SUBAPPLICATION Uebung_011f_AX (* Numeric Value Input I3 Durchschleifen auf N3 (Input und Output PHYS via NumericObjectPool_S) *)
  (* Standard: 61499-2; Description: Copyright (c) 2023 Meisterschulen am Ostbahnhof This program and the accompanying materials are made available under the terms of the Eclipse Public License 2.0 which is available at https://www.eclipse.org/legal/epl-2.0/ SPDX-License-Identifier: EPL-2.0 *)
  (* Version 1.0, 2026-04-14, Franz Höpfinger, Meisterschulen am Ostbahnhof, initial API and implementation and/or initial documentation *)
  PACKAGE Uebungen;
  IMPORT Uebungen::const::UT::DefaultPool_Numeric::InputNumber_I3_N;
  IMPORT Uebungen::const::UT::DefaultPool_Numeric::OutputNumber_N3_N;
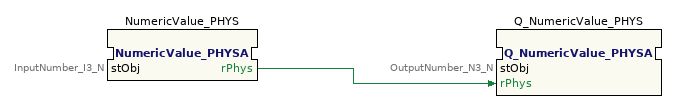
  (* Beispiel: I3-Eingabe -500.00 → rPhys=-500.0 → Q_NumericValue_PHYS(N3) → N3 zeigt -500.00. *)
  FBS
    NumericValue_PHYS : isobus::UT::io::NumericValue::NumericValue_PHYSA(stObj := InputNumber_I3_N);
    Q_NumericValue_PHYS : isobus::UT::Q::Q_NumericValue_PHYSA(stObj := OutputNumber_N3_N);
  END_FBS
  ADAPTER_CONNECTIONS
    NumericValue_PHYS.rPhys TO Q_NumericValue_PHYS.rPhys;
  END_CONNECTIONS
END_SUBAPPLICATION
